TYPE E_ChargerState :
(
    Idle := 0,
    ModulesOff := 10,
    SetVI := 20,
    CheckVoltage := 30,
    EnableModules := 40,
    Running := 100,
    Shutdown := 200,
    OpenRelay := 210,
    Fault := 900
);
END_TYPE

(* stored: Version 1.1.0.1, ProductVersion 3.1.4026.18
   DUT E_ChargerState: Id {73d979d3-002a-43e6-8b13-29ff42e14b6f} *)
